{attribute 'qualified_only'}
{attribute 'strict'}
{attribute 'to_string'}
TYPE EBufferStatus :
(
	Leeg := 0,
	Vol,
	Error
);
END_TYPE

(* stored: Version 1.1.0.1
   DUT EBufferStatus: Id {9ed94363-c354-4a3b-97f9-de3966a61e0a} *)
